// TIA Portal V17 export
// export: Created 2024-09-02T12:50:30.2505606Z, ExportSetting WithDefaults, DisplayName Totally Integrated Automation Portal, DisplayVersion V17, DisplayName TIA Portal Openness, DisplayVersion V17, DisplayName TIA Portal Version Control Interface, DisplayVersion V17, DisplayName STEP 7 Professional, DisplayVersion V17, DisplayName STEP 7 Safety, DisplayVersion V17, DisplayName WinCC Professional, DisplayVersion V17
TYPE "type_CognexDMin"
// stored: IsFailsafeCompliant false
   STRUCT
      Status { ExternalWritable := 'False'} : Struct
         Trigger_Ready { ExternalWritable := 'False'} : Bool;   // Aufnahmestatus: Trigger Ready / Recording status: Trigger Ready
         Trigger_Ack { ExternalWritable := 'False'} : Bool;   // Aufnahmestatus: Trigger Acknowledge / Recording status: Trigger Acknowledge
         Acquiring { ExternalWritable := 'False'} : Bool;   // Aufnahmestatus: Acquiring / Recording Status: Acquiring
         Missed_Ack { ExternalWritable := 'False'} : Bool;   // Aufnahmestatus: Missed Acknowledge / Recording Status: Missed Acknowledge
         Offline_Reason_0 { ExternalWritable := 'False'} : Bool;   // Aufnahmestatus: Offline Reason Bit 0 / Recording status: Offline Reason Bit 0
         Offline_Reason_1 { ExternalWritable := 'False'} : Bool;   // Aufnahmestatus: Offline Reason Bit 1 / Recording status: Offline Reason Bit 1
         Offline_Reason_2 { ExternalWritable := 'False'} : Bool;   // Aufnahmestatus: Offline Reason Bit 2 / Recording status: Offline Reason Bit 2
         Online { ExternalWritable := 'False'} : Bool;   // Aufnahmestatus: Online / Recording status: Online
         TriggerIDhi { ExternalWritable := 'False'} : Byte;   // Aufnahmestatus: Acquiring ID Hi / Recording Status: Acquiring ID Hi
         TriggerIDlo { ExternalWritable := 'False'} : Byte;   // Aufnahmestatus: Acquiring ID Lo / Recording Status: Acquiring ID Lo
         Decoding { ExternalWritable := 'False'} : Bool;   // Inspektionsstatus: Inspecting / Inspection Status: Inspecting
         Decoding_complete { ExternalWritable := 'False'} : Bool;   // Inspektionsstatus: Inspection Complete / Inspection status: Inspection Complete
         Results_Buffer_Overrun { ExternalWritable := 'False'} : Bool;   // Inspektionsstatus: Results Buffer Overrung / Inspection Status: Results Buffer Overrung
         Results_Available { ExternalWritable := 'False'} : Bool;   // Inspektionsstatus: Results Valid / Inspection Status: Results Valid
         Job_loading { ExternalWritable := 'False'} : Bool;   // Inspektionsstatus: Job Loading / Inspection Status: Job Loading
         Job_load_complete { ExternalWritable := 'False'} : Bool;   // Inspektionsstatus: Job Load Complete / Inspection Status: Job Load Complete
         Job_load_failed { ExternalWritable := 'False'} : Bool;   // Inspektionsstatus: Job Load Failed / Inspection Status: Job Load Failed
         General_Fault { ExternalWritable := 'False'} : Bool;   // Inspektionsstatus: Fault / Inspection status: Fault
         Job_No { ExternalWritable := 'False'} : Byte;   // Parametersatz: Job Number / Parameter set: Job Number
         Softevent { ExternalWritable := 'False'} : Byte;   // Softevent / soft event
      END_STRUCT;
      Ergebnissdaten { ExternalWritable := 'False'} : Struct   // User Daten / User data
         Result { ExternalWritable := 'False'} : Struct   // Option
            ID { ExternalWritable := 'False'} : Int;   // Kennung für die Ausführungsart des IBV-Systems / Identifier for the type of implementation of the IBV system
            Code { ExternalWritable := 'False'} : Int;   // Aktuelle Modis: TR-> Bildaufnahme und -auswertung durchführen / Current modes: TR-> Perform image acquisition and evaluation
            Extendet { ExternalWritable := 'False'} : Int;
            Length { ExternalWritable := 'False'} : Int;
         END_STRUCT;
         Data { ExternalWritable := 'False'} : Struct
            Data { ExternalWritable := 'False'} : Array[1..246] of Char;   // User Daten / User data
         END_STRUCT;
      END_STRUCT;
   END_STRUCT;
END_TYPE
